// TIA Portal V20 export
TYPE "typeSyncNode"
TITLE = typeEquipmentC_SyncNode
// Module synchronous control nodes including synchronous control nodes from child modules
// stored: Namespace Unit1.Em1
   STRUCT
      commands { ExternalWritable := 'False'} : Struct   // Example of commands. Must be adjusted depending on the application.
         enableHpMotion : Bool;   // Enable High performance motion program
      END_STRUCT;
      status { ExternalWritable := 'False'} : Struct   // Example of status bits. Must be adjusted depending on the application.
         busy : Bool;   // Logic that is executed in the motion cycle is busy
         error : Bool;   // Logic that is executed in the motion cycle has an error
      END_STRUCT;
      WinderInput { S7_SetPoint := 'True'} : "LConSMC_typeWinderInput";
      WinderOutput { S7_SetPoint := 'True'} : "LConSMC_typeWinderOutput";
      WinderConfig { S7_SetPoint := 'True'} : "LConSMC_typeWinderConfig";
      WinderDiag { S7_SetPoint := 'True'} : "LConSMC_typeWinderDiag";
   END_STRUCT;
END_TYPE
